DECL PDAT PPDAT62={VEL 100.000,ACC 100.000,APO_DIST 100.000,GEAR_JERK 50.0000,EXAX_IGN 3}
DECL E6POS XP88={X 1141.74707,Y -756.804688,Z 1738.58630,A -3.18880939,B -12.7060452,C -88.0300903,S 2,T 42,E1 193.394,E2 193.959457,E3 193.454041,E4 0.0,E5 0.0,E6 0.0}
DECL FDAT FP88={TOOL_NO 1,BASE_NO 0,IPO_FRAME #BASE,POINT2[] " ",TQ_STATE FALSE}
DECL PDAT PPDAT63={VEL 100.000,ACC 100.000,APO_DIST 100.000,GEAR_JERK 50.0000,EXAX_IGN 3}
DECL E6POS XP89={X 1142.69055,Y -830.857117,Z 1649.52417,A -10.4538889,B -8.34854698,C -156.497650,S 2,T 10,E1 193.394,E2 193.959457,E3 193.454041,E4 0.0,E5 0.0,E6 0.0}
DECL FDAT FP89={TOOL_NO 1,BASE_NO 0,IPO_FRAME #BASE,POINT2[] " ",TQ_STATE FALSE}
DECL PDAT PPDAT64={VEL 100.000,ACC 100.000,APO_DIST 100.000,GEAR_JERK 50.0000,EXAX_IGN 3}
DECL E6POS XP90={X 1195.77185,Y -873.118225,Z 1662.25977,A -14.0592203,B 6.95337057,C -34.2239,S 2,T 42,E1 193.394,E2 193.959457,E3 193.454041,E4 0.0,E5 0.0,E6 0.0}
DECL FDAT FP90={TOOL_NO 1,BASE_NO 0,IPO_FRAME #BASE,POINT2[] " ",TQ_STATE FALSE}
DECL PDAT PPDAT65={VEL 100.000,ACC 100.000,APO_DIST 100.000,GEAR_JERK 50.0000,EXAX_IGN 3}
DECL LDAT LCPDAT28={ACC 100.000,APO_DIST 100.000,APO_FAC 50.0000,AXIS_VEL 100.000,AXIS_ACC 100.000,ORI_TYP #VAR,CIRC_TYP #BASE,JERK_FAC 50.0000,GEAR_JERK 50.0000,EXAX_IGN 0}
DECL PDAT PPDAT66={ACC 100.000,APO_DIST 100.000,APO_MODE #CPTP,GEAR_JERK 50.0000}
DECL E6POS XP91={X 1061.26965,Y -789.098206,Z 1693.26929,A -9.41882229,B 13.6831732,C 140.354233,S 2,T 42,E1 54.1421051,E2 193.959457,E3 193.453949,E4 0.0,E5 0.0,E6 0.0}
DECL FDAT FP91={TOOL_NO 1,BASE_NO 0,IPO_FRAME #BASE,POINT2[] " ",TQ_STATE FALSE}
DECL PDAT PPDAT67={VEL 100.000,ACC 100.000,APO_DIST 100.000,GEAR_JERK 50.0000,EXAX_IGN 3}
DECL E6POS XP92={X 1153.79370,Y -796.864563,Z 1655.69360,A 2.99197602,B 13.8469086,C 102.009964,S 2,T 42,E1 63.9584465,E2 193.959412,E3 193.453964,E4 0.0,E5 0.0,E6 0.0}
DECL FDAT FP92={TOOL_NO 1,BASE_NO 0,IPO_FRAME #BASE,POINT2[] " ",TQ_STATE FALSE}
DECL PDAT PPDAT68={VEL 100.000,ACC 100.000,APO_DIST 100.000,GEAR_JERK 50.0000,EXAX_IGN 3}
DECL E6POS XP93={X 1178.07373,Y -747.549744,Z 1629.13306,A 5.99540949,B 16.6131,C 102.466103,S 2,T 42,E1 63.9584656,E2 193.959412,E3 193.453964,E4 0.0,E5 0.0,E6 0.0}
DECL FDAT FP93={TOOL_NO 1,BASE_NO 0,IPO_FRAME #BASE,POINT2[] " ",TQ_STATE FALSE}
DECL PDAT PPDAT69={VEL 100.000,ACC 100.000,APO_DIST 100.000,GEAR_JERK 50.0000,EXAX_IGN 3}
DECL E6POS XP94={X 1323.82373,Y -609.951843,Z 1568.18591,A 14.6684265,B 18.8945389,C 101.399376,S 2,T 42,E1 63.9584923,E2 193.959412,E3 193.453964,E4 0.0,E5 0.0,E6 0.0}
DECL FDAT FP94={TOOL_NO 1,BASE_NO 0,IPO_FRAME #BASE,POINT2[] " ",TQ_STATE FALSE}
DECL PDAT PPDAT70={VEL 100.000,ACC 100.000,APO_DIST 100.000,GEAR_JERK 50.0000,EXAX_IGN 3}
DECL E6POS XP95={X 1320.98547,Y -625.368042,Z 1554.23413,A 14.7803907,B 20.3776741,C 99.3829498,S 2,T 42,E1 63.9585266,E2 193.959412,E3 193.453964,E4 0.0,E5 0.0,E6 0.0}
DECL FDAT FP95={TOOL_NO 1,BASE_NO 0,IPO_FRAME #BASE,POINT2[] " ",TQ_STATE FALSE}
DECL PDAT PPDAT71={VEL 100.000,ACC 100.000,APO_DIST 100.000,GEAR_JERK 50.0000,EXAX_IGN 3}
DECL E6POS XP96={X 1041.34229,Y -292.671356,Z 1868.38,A 20.5019817,B 9.28383160,C 88.9917,S 2,T 42,E1 63.9585266,E2 193.959412,E3 193.453964,E4 0.0,E5 0.0,E6 0.0}
DECL FDAT FP96={TOOL_NO 1,BASE_NO 0,IPO_FRAME #BASE,POINT2[] " ",TQ_STATE FALSE}
DECL PDAT PPDAT72={VEL 100.000,ACC 100.000,APO_DIST 100.000,GEAR_JERK 50.0000,EXAX_IGN 3}
DECL E6POS XP97={X 1299.18445,Y -307.536926,Z 1659.69568,A 25.6714821,B 17.5003357,C 89.9028168,S 2,T 42,E1 63.9585266,E2 193.959412,E3 193.453964,E4 0.0,E5 0.0,E6 0.0}
DECL FDAT FP97={TOOL_NO 1,BASE_NO 0,IPO_FRAME #BASE,POINT2[] " ",TQ_STATE FALSE}
DECL PDAT PPDAT73={VEL 100.000,ACC 100.000,APO_DIST 100.000,GEAR_JERK 50.0000,EXAX_IGN 3}
DECL E6POS XP98={X 1398.85815,Y -242.372314,Z 1593.69446,A 29.9672890,B 18.8260975,C 84.7787704,S 2,T 42,E1 63.9585266,E2 193.959412,E3 193.453964,E4 0.0,E5 0.0,E6 0.0}
DECL FDAT FP98={TOOL_NO 1,BASE_NO 0,IPO_FRAME #BASE,POINT2[] " ",TQ_STATE FALSE}
DECL PDAT PPDAT74={VEL 100.000,ACC 100.000,APO_DIST 100.000,GEAR_JERK 50.0000,EXAX_IGN 3}
DECL E6POS XP99={X 1417.56384,Y -77.8548,Z 1593.69446,A 36.6534042,B 18.8260975,C 84.7787704,S 2,T 42,E1 63.9585266,E2 193.959412,E3 193.453964,E4 0.0,E5 0.0,E6 0.0}
DECL FDAT FP99={TOOL_NO 1,BASE_NO 0,IPO_FRAME #BASE,POINT2[] " ",TQ_STATE FALSE}
DECL PDAT PPDAT75={VEL 100.000,ACC 100.000,APO_DIST 100.000,GEAR_JERK 50.0000,EXAX_IGN 3}
DECL E6POS XP100={X 1441.90417,Y -8.89344883,Z 1568.05261,A 46.5573349,B 22.9023724,C 70.7657547,S 2,T 42,E1 63.9585266,E2 193.959412,E3 193.453964,E4 0.0,E5 0.0,E6 0.0}
DECL FDAT FP100={TOOL_NO 1,BASE_NO 0,IPO_FRAME #BASE,POINT2[] " ",TQ_STATE FALSE}
DECL PDAT PPDAT76={VEL 100.000,ACC 100.000,APO_DIST 100.000,GEAR_JERK 50.0000,EXAX_IGN 3}
DECL E6POS XP101={X 1273.96033,Y 11.5089941,Z 1695.40906,A 45.3334694,B 20.0161724,C 67.0416183,S 2,T 42,E1 63.9585266,E2 193.959412,E3 193.453964,E4 0.0,E5 0.0,E6 0.0}
DECL FDAT FP101={TOOL_NO 1,BASE_NO 0,IPO_FRAME #BASE,POINT2[] " ",TQ_STATE FALSE}
DECL PDAT PPDAT77={VEL 100.000,ACC 100.000,APO_DIST 100.000,GEAR_JERK 50.0000,EXAX_IGN 3}
DECL E6POS XP102={X 1139.76379,Y 336.898346,Z 1800.55127,A 54.9098129,B 11.6087036,C 61.9939919,S 2,T 43,E1 63.9585266,E2 193.959412,E3 193.453964,E4 0.0,E5 0.0,E6 0.0}
DECL FDAT FP102={TOOL_NO 1,BASE_NO 0,IPO_FRAME #BASE,POINT2[] " ",TQ_STATE FALSE}
DECL PDAT PPDAT78={VEL 100.000,ACC 100.000,APO_DIST 100.000,GEAR_JERK 50.0000,EXAX_IGN 3}
DECL E6POS XP103={X 1354.29443,Y 51.7001877,Z 1702.54919,A 35.0817719,B -8.09186363,C 89.4801788,S 2,T 42,E1 -0.571967244,E2 193.829330,E3 193.453964,E4 0.0,E5 0.0,E6 0.0}
DECL FDAT FP103={TOOL_NO 1,BASE_NO 0,IPO_FRAME #BASE,POINT2[] " ",TQ_STATE FALSE}
DECL PDAT PPDAT79={VEL 100.000,ACC 100.000,APO_DIST 100.000,GEAR_JERK 50.0000,EXAX_IGN 3}
DECL E6POS XP104={X 1385.38855,Y -220.764191,Z 1641.26550,A 24.4803696,B -4.30105639,C 89.7629471,S 2,T 42,E1 -0.571967244,E2 193.829330,E3 193.453964,E4 0.0,E5 0.0,E6 0.0}
DECL FDAT FP104={TOOL_NO 1,BASE_NO 0,IPO_FRAME #BASE,POINT2[] " ",TQ_STATE FALSE}
DECL PDAT PPDAT80={VEL 100.000,ACC 100.000,APO_DIST 100.000,GEAR_JERK 50.0000,EXAX_IGN 3}
DECL E6POS XP105={X 1289.38306,Y -252.188782,Z 1731.30444,A 22.5847874,B -7.73033381,C 86.7184830,S 2,T 42,E1 -0.571967244,E2 193.829330,E3 193.453964,E4 0.0,E5 0.0,E6 0.0}
DECL FDAT FP105={TOOL_NO 1,BASE_NO 0,IPO_FRAME #BASE,POINT2[] " ",TQ_STATE FALSE}
DECL PDAT PPDAT81={VEL 100.000,ACC 100.000,APO_DIST 100.000,GEAR_JERK 50.0000,EXAX_IGN 3}
DECL E6POS XP106={X 1257.58044,Y -896.735657,Z 1551.46667,A 12.9449339,B 8.12423706,C 75.5191879,S 2,T 42,E1 -0.571962535,E2 193.829300,E3 193.453934,E4 0.0,E5 0.0,E6 0.0}
DECL FDAT FP106={TOOL_NO 1,BASE_NO 0,IPO_FRAME #BASE,POINT2[] " ",TQ_STATE FALSE}
DECL PDAT PPDAT82={VEL 100.000,ACC 100.000,APO_DIST 100.000,GEAR_JERK 50.0000,EXAX_IGN 3}
DECL E6POS XP107={X 1229.18567,Y 245.689148,Z 1812.89673,A 16.9957695,B 12.3257923,C 12.0421877,S 2,T 43,E1 193.394104,E2 193.959641,E3 193.454254,E4 0.0,E5 0.0,E6 0.0}
DECL FDAT FP107={TOOL_NO 1,BASE_NO 0,IPO_FRAME #BASE,POINT2[] " ",TQ_STATE FALSE}
DECL PDAT PPDAT83={VEL 100.000,ACC 100.000,APO_DIST 100.000,GEAR_JERK 50.0000,EXAX_IGN 3}
DECL E6POS XP108={X 1429.67847,Y 345.693054,Z 1603.58435,A 54.0950737,B 16.8773441,C 68.3533478,S 2,T 43,E1 63.9585266,E2 193.959412,E3 193.453964,E4 0.0,E5 0.0,E6 0.0}
DECL FDAT FP108={TOOL_NO 1,BASE_NO 0,IPO_FRAME #BASE,POINT2[] " ",TQ_STATE FALSE}
DECL PDAT PPDAT84={VEL 100.000,ACC 100.000,APO_DIST 100.000,GEAR_JERK 50.0000,EXAX_IGN 3}
DECL E6POS XP109={X 1404.29797,Y 376.847015,Z 1637.55579,A 45.0448,B -10.3995733,C 96.5909729,S 2,T 43,E1 2.07479143,E2 193.834671,E3 193.453964,E4 0.0,E5 0.0,E6 0.0}
DECL FDAT FP109={TOOL_NO 1,BASE_NO 0,IPO_FRAME #BASE,POINT2[] " ",TQ_STATE FALSE}
DECL PDAT PPDAT85={VEL 100.000,ACC 100.000,APO_DIST 100.000,GEAR_JERK 50.0000,EXAX_IGN 3}
ENDDAT
